FUNCTION_BLOCK REAL_Param
VAR_INPUT PERSISTENT
	val			: REAL;
END_VAR

END_FUNCTION_BLOCK

(* stored: Version 1.1.0.1
   POU REAL_Param: Id {c5204730-3360-4f94-a588-83d0bfaa453c}, SpecialFunc None *)
